	                    #sFB_Conveyor330(iUDT_ConveyorConfiguration := #iUDT_Configuration."330".Conveyor,
	                                     idi_PECEoSDistance := #iUDT_Configuration."330".PEC_Eos.Distance,
	                                     idi_PECBoSDistance := 0,
	                                     ii_ExternalSpeed := 0,
	                                     ix_SafetyOk := #ix_SafetyOk,
	                                     ix_24vOk := #ix_24vOk,
	                                     ix_400vOk := #ix_400vOk,
	                                     ix_HardwareOk := #ix_HardwareOk,
	                                     ix_PECEoS := #iqUDT_WorkstationStatus."330".PEC_EoS.PEC,
	                                     ix_PECBoS := TRUE,
	                                     ix_ReverseDirection := FALSE,
	                                     ix_ExternalRequestDieBack := FALSE,
	                                     ix_ExternalRequestHold := #sx_LeftExternalRequestHold330,
	                                     ix_ResetEnergySave := FALSE,
	                                     qUDT_HMIStatus => #iqUDT_WorkstationStatus."330".Conveyor,
	                                     qUDT_Status => #iqUDT_WorkstationCommonStatus."330",
	                                     iqUDT_EquipmentControl := #iqUDT_EquipmentControl,
	                                     iqUDT_ConveyorCommand := #iqUDT_WorkstationCommands."330".Conveyor,
	                                     iqUDT_ConveyorInterface := #sUDT_Interface330,
	                                     iqUDT_HandShakeUp := #sUDT_Handshake320,
	                                     iqUDT_HandShake := #sUDT_Handshake330,
	                                     iqUDT_Statistics := #iqUDT_WorkstationStatistics."330".Conveyor);
	                END_REGION

	                REGION MCO

	                    #sFB_MCOConveyLinxAixController330(iUDT_AixConfig := #iUDT_Configuration."330".MCO_M01,
	                                                       iUDT_AixInputsModule := #iUDT_MotorInput330,
	                                                       ix_24vOk := #ix_24vOk,
	                                                       ix_SimulationModeActive := "DB_Memory".Simulation,
	                                                       ii_MotorPositionId := 1,
	                                                       qUDT_HMIStatus => #iqUDT_WorkstationStatus."330".MCO_M01,
	                                                       iqUDT_AixOutputsModule := #iqUDT_MotorOutput330,
	                                                       iqUDT_ConveyorInterface := #sUDT_Interface330,
	                                                       iqUDT_MCOStatistics := #iqUDT_WorkstationStatistics."330".MCO_M01);
	                END_REGION
	            END_REGION

	            REGION 340

	                REGION Displacement

	                    #sFB_Displacement340(#sUDT_Interface340);

	                END_REGION

	                REGION EOS
	                    #sFB_PEC340(ix_PEC := NOT #iUDT_MotorInput330.AllSensorPortInputs.RightSensor,
	                                iUDT_PECConfiguration := #iUDT_Configuration."340".PEC_Eos,
	                                qx_PECFiltered => #tx_dummy,
	                                qUDT_HMIStatus => #iqUDT_WorkstationStatus."340".PEC_EoS,
	                                iqUDT_ConveyorInterface := #sUDT_Interface340,
	                                iqUDT_PECStatistics := #iqUDT_WorkstationStatistics."340".PEC_EoS);


	                END_REGION


	                REGION Conveyor

	                    #sFB_Conveyor340(iUDT_ConveyorConfiguration := #iUDT_Configuration."340".Conveyor,
	                                     idi_PECEoSDistance := #iUDT_Configuration."340".PEC_Eos.Distance,
	                                     idi_PECBoSDistance := 0,
	                                     ii_ExternalSpeed := 0,
	                                     ix_SafetyOk := #ix_SafetyOk,
	                                     ix_24vOk := #ix_24vOk,
	                                     ix_400vOk := #ix_400vOk,
	                                     ix_HardwareOk := #ix_HardwareOk,
	                                     ix_PECEoS := #iqUDT_WorkstationStatus."340".PEC_EoS.PEC,
	                                     ix_PECBoS := TRUE,
	                                     ix_ReverseDirection := FALSE,
	                                     ix_ExternalRequestDieBack := FALSE,
	                                     ix_ExternalRequestHold := #sx_LeftExternalRequestHold340,
	                                     ix_ResetEnergySave := FALSE,
	                                     qUDT_HMIStatus => #iqUDT_WorkstationStatus."340".Conveyor,
	                                     qUDT_Status => #iqUDT_WorkstationCommonStatus."340",
	                                     iqUDT_EquipmentControl := #iqUDT_EquipmentControl,
	                                     iqUDT_ConveyorCommand := #iqUDT_WorkstationCommands."340".Conveyor,
	                                     iqUDT_ConveyorInterface := #sUDT_Interface340,
	                                     iqUDT_HandShakeUp := #sUDT_Handshake330,
	                                     iqUDT_HandShake := #sUDT_Handshake340,
	                                     iqUDT_Statistics := #iqUDT_WorkstationStatistics."340".Conveyor);
	                END_REGION

	                REGION MCO

	                    #sFB_MCOConveyLinxAixController340(iUDT_AixConfig := #iUDT_Configuration."340".MCO_M01,
	                                                       iUDT_AixInputsModule := #iUDT_MotorInput330,
	                                                       ix_24vOk := #ix_24vOk,
	                                                       ix_SimulationModeActive := "DB_Memory".Simulation,
	                                                       ii_MotorPositionId := 2,
	                                                       qUDT_HMIStatus => #iqUDT_WorkstationStatus."340".MCO_M01,
	                                                       iqUDT_AixOutputsModule := #iqUDT_MotorOutput330,
	                                                       iqUDT_ConveyorInterface := #sUDT_Interface340,
	                                                       iqUDT_MCOStatistics := #iqUDT_WorkstationStatistics."340".MCO_M01);
	                END_REGION
	            END_REGION

	            REGION 350

	                REGION Displacement

	                    #sFB_Displacement350(#sUDT_Interface350);

	                END_REGION

	                REGION EOS
	                    #sFB_PEC350(ix_PEC := NOT #iUDT_MotorInput350.AllSensorPortInputs.LeftSensor,
	                                iUDT_PECConfiguration := #iUDT_Configuration."350".PEC_Eos,
	                                qx_PECFiltered => #tx_dummy,
	                                qUDT_HMIStatus => #iqUDT_WorkstationStatus."350".PEC_EoS,
	                                iqUDT_ConveyorInterface := #sUDT_Interface350,
	                                iqUDT_PECStatistics := #iqUDT_WorkstationStatistics."350".PEC_EoS);

	                END_REGION

	                REGION Conveyor

	                    #sUDT_Handshake350.RTR := #sUDT_Handshake350.RTR OR #iqUDT_WorkstationStatus."350".PEC_EoS.PEC;

	                    #sFB_Conveyor350(iUDT_ConveyorConfiguration := #iUDT_Configuration."350".Conveyor,
	                                     idi_PECEoSDistance := #iUDT_Configuration."350".PEC_Eos.Distance,
	                                     idi_PECBoSDistance := 0,
	                                     ii_ExternalSpeed := 0,
	                                     ix_SafetyOk := #ix_SafetyOk,
	                                     ix_24vOk := #ix_24vOk,
	                                     ix_400vOk := #ix_400vOk,
	                                     ix_HardwareOk := #ix_HardwareOk,
	                                     ix_PECEoS := #iqUDT_WorkstationStatus."350".PEC_EoS.PEC,
	                                     ix_PECBoS := TRUE,
	                                     ix_ReverseDirection := FALSE,
	                                     ix_ExternalRequestDieBack := FALSE,
	                                     ix_ExternalRequestHold := #sx_LeftExternalRequestHold350,
	                                     ix_ResetEnergySave := FALSE,
	                                     qUDT_HMIStatus => #iqUDT_WorkstationStatus."350".Conveyor,
	                                     qUDT_Status => #iqUDT_WorkstationCommonStatus."350",
	                                     iqUDT_EquipmentControl := #iqUDT_EquipmentControl,
	                                     iqUDT_ConveyorCommand := #iqUDT_WorkstationCommands."350".Conveyor,
	                                     iqUDT_ConveyorInterface := #sUDT_Interface350,
	                                     iqUDT_HandShakeUp := #sUDT_Handshake340,
	                                     iqUDT_HandShake := #sUDT_Handshake350,
	                                     iqUDT_Statistics := #iqUDT_WorkstationStatistics."350".Conveyor);
	                END_REGION

	                REGION MCO

	                    #sFB_MCOConveyLinxAixController350(iUDT_AixConfig := #iUDT_Configuration."350".MCO_M01,
	                                                       iUDT_AixInputsModule := #iUDT_MotorInput350,
	                                                       ix_24vOk := #ix_24vOk,
	                                                       ix_SimulationModeActive := "DB_Memory".Simulation,
	                                                       ii_MotorPositionId := 1,
	                                                       qUDT_HMIStatus => #iqUDT_WorkstationStatus."350".MCO_M01,
	                                                       iqUDT_AixOutputsModule := #iqUDT_MotorOutput350,
	                                                       iqUDT_ConveyorInterface := #sUDT_Interface350,
	                                                       iqUDT_MCOStatistics := #iqUDT_WorkstationStatistics."350".MCO_M01);
	                END_REGION
	            END_REGION
	        END_REGION
	    END_IF;
	END_REGION

	REGION 6 - Right station
	    IF #iUDT_Configuration.GlobalConfig.RightStationExists THEN

	        REGION 6.1 - Indexing

	            // Start indexing after request if there are empty stations and no pushout is active
	            IF #iqUDT_CommunicationWES.RightWorkstation.StartIndexing AND #si_RightEmptyStations > 0
	                AND NOT (#sx_RightPushOutActiveStation1
	                OR #sx_RightPushOutActiveStation2
	                OR #sx_RightPushOutActiveStation3
	                OR #sx_RightPushOutActiveStation4
	                OR #sx_RightPushOutActiveStation5) THEN

	                #sx_RightIndexing := TRUE;
	            END_IF;

	            IF NOT #sx_RightIndexing THEN                                      // If there is no indexing in progress

	                #si_RightDestinationC541 := 0;                                // Reset RAT destination
	                #sx_RightExternalRequestHold550 := TRUE;                      // Hold station conveyors
	                #sx_RightExternalRequestHold560 := TRUE;
	                #sx_RightExternalRequestHold570 := TRUE;
	                #sx_RightExternalRequestHold580 := TRUE;
	                #sx_RightExternalRequestHold590 := TRUE;

	            ELSE

	                IF #sR_TRIG_PEC540.Q AND #si_RightEmptyStations > 0 THEN       //Count down empty stations after diverting a tote into station
	                    #si_RightEmptyStations -= 1;
	                END_IF;

	                #si_RightDestinationC541 := 1;                               // Set RAT destination
	                #sx_RightExternalRequestHold550 := FALSE;                    // Release hold of station conveyors
	                #sx_RightExternalRequestHold560 := FALSE;
	                #sx_RightExternalRequestHold570 := FALSE;
	                #sx_RightExternalRequestHold580 := FALSE;
	                #sx_RightExternalRequestHold590 := FALSE;

	                IF                                                           //End indexing when all totes are on position
	                    NOT #iqUDT_WorkstationStatus."550".PEC_EoS.PEC
	                    AND NOT #iqUDT_WorkstationStatus."560".PEC_EoS.PEC
	                    AND NOT #iqUDT_WorkstationStatus."570".PEC_EoS.PEC
	                    AND NOT #iqUDT_WorkstationStatus."580".PEC_EoS.PEC
	                    AND NOT #iqUDT_WorkstationStatus."590".PEC_EoS.PEC
	                    AND NOT (#sUDT_Interface550.ActualSpeed > 0) THEN

	                    #sx_RightIndexing := FALSE;

	                END_IF;
	            END_IF;

	        END_REGION

	        REGION 6.2 - Push Out

	            REGION 6.2.0 - Pushout conveyors hold
	                IF #sFB_TimerOnOffDelay_Hold710.qx_DelayedSignal THEN
	                    #sx_RightExternalRequestHold710 := TRUE;
	                END_IF;

	                IF #sFB_TimerOnOffDelay_Hold720.qx_DelayedSignal THEN
	                    #sx_RightExternalRequestHold720 := TRUE;
	                END_IF;

	                IF #sFB_TimerOnOffDelay_Hold730.qx_DelayedSignal THEN
	                    #sx_RightExternalRequestHold730 := TRUE;
	                END_IF;

	                IF #sFB_TimerOnOffDelay_Hold740.qx_DelayedSignal THEN
	                    #sx_RightExternalRequestHold740 := TRUE;
	                END_IF;

	                IF #sFB_TimerOnOffDelay_Hold750.qx_DelayedSignal THEN
	                    #sx_RightExternalRequestHold750 := TRUE;
	                END_IF;
	            END_REGION

	            REGION 6.2.1 - Push Out Station 1

	                // Start automatic pushout after request if there is no indexing procedure and a tote is present on first station
	                IF #iqUDT_CommunicationWES.RightWorkstation.Station1.ReadyForPush AND NOT #sx_RightIndexing
	                    AND NOT #iqUDT_WorkstationStatus."590".PEC_EoS.PEC THEN

	                    #sx_RightPushOutActiveStation1 := TRUE;
	                END_IF;

	                IF #sx_RightPushOutActiveStation1 THEN                         //release hold
	                    #sx_RightExternalRequestHold590 := FALSE;

	                    IF #sFB_RightAngledTransfer611.qx_ExternalSendRequestB THEN    //after tote is already on RAT, hold the conveyor and end pushout procedure
	                        #sx_RightExternalRequestHold590 := TRUE;
	                        #sx_RightPushOutActiveStation1 := FALSE;
	                    END_IF;
	                END_IF;

	            END_REGION

	            REGION 6.2.2 - Push Out station 2

	                IF #iqUDT_CommunicationWES.RightWorkstation.Station2.ReadyForPush THEN        //set pushout to active after request
	                    #sx_RightPushOutActiveStation2 := TRUE;
	                END_IF;

	                IF #sx_RightPushOutActiveStation2                               // After station is empty and tote has been detected on pushout conveyor release holds
	                    AND #iqUDT_WorkstationStatus."580".PEC_EoS.PEC
	                    AND #sFB_TimerOnOffDelay_Detect740.qx_DelayedSignal THEN

	                    #sx_RightExternalRequestHold740 := FALSE;
	                    #sx_RightExternalRequestHold750 := FALSE;

	                    FILL_BLK(IN := 0,                                             //clear tracking
	                             COUNT := REAL_TO_ULINT(DINT_TO_REAL(#iUDT_Configuration."580".Conveyor.Common.Length) * #cr_ClearTrackingModifier),
	                             OUT => #sa_TrackingArray580[0]);

	                    #sx_RightPushOutActiveStation2 := FALSE;                       //end pushout procedure

	                END_IF;


	            END_REGION

	            REGION 6.2.3 - Push Out station 3

	                IF #iqUDT_CommunicationWES.RightWorkstation.Station3.ReadyForPush THEN          //set pushout to active after request
	                    #sx_RightPushOutActiveStation3 := TRUE;
	                END_IF;

	                IF #sx_RightPushOutActiveStation3
	                    AND #iqUDT_WorkstationStatus."570".PEC_EoS.PEC
	                    AND #sFB_TimerOnOffDelay_Detect730.qx_DelayedSignal THEN                // After station is empty and tote has been detected on pushout conveyor release holds

	                    #sx_RightExternalRequestHold730 := FALSE;
	                    #sx_RightExternalRequestHold740 := FALSE;
	                    #sx_RightExternalRequestHold750 := FALSE;

	                    FILL_BLK(IN := 0,                                                         //clear tracking
	                             COUNT := REAL_TO_ULINT(DINT_TO_REAL(#iUDT_Configuration."570".Conveyor.Common.Length) * #cr_ClearTrackingModifier),
	                             OUT => #sa_TrackingArray570[0]);

	                    #sx_RightPushOutActiveStation3 := FALSE;                              //end pushout procedure

	                END_IF;
	            END_REGION

	            REGION 6.2.4 - Push Out station 4

	                IF #iqUDT_CommunicationWES.RightWorkstation.Station4.ReadyForPush THEN              //set pushout to active after request
	                    #sx_RightPushOutActiveStation4 := TRUE;
	                END_IF;

	                IF #sx_RightPushOutActiveStation4
	                    AND #iqUDT_WorkstationStatus."560".PEC_EoS.PEC
	                    AND #sFB_TimerOnOffDelay_Detect720.qx_DelayedSignal THEN                // After station is empty and tote has been detected on pushout conveyor release holds

	                    #sx_RightExternalRequestHold720 := FALSE;
	                    #sx_RightExternalRequestHold730 := FALSE;
	                    #sx_RightExternalRequestHold740 := FALSE;
	                    #sx_RightExternalRequestHold750 := FALSE;

	                    FILL_BLK(IN := 0,                                                      //clear tracking
	                             COUNT := REAL_TO_ULINT(DINT_TO_REAL(#iUDT_Configuration."560".Conveyor.Common.Length) * #cr_ClearTrackingModifier),
	                             OUT => #sa_TrackingArray560[0]);

	                    #sx_RightPushOutActiveStation4 := FALSE;                          //end pushout procedure

	                END_IF;

	            END_REGION

	            REGION 6.2.5 - Push Out station 5

	                IF #iqUDT_CommunicationWES.RightWorkstation.Station5.ReadyForPush THEN          //set pushout to active after request
	                    #sx_RightPushOutActiveStation5 := TRUE;
	                END_IF;

	                IF #sx_RightPushOutActiveStation5
	                    AND #iqUDT_WorkstationStatus."550".PEC_EoS.PEC
	                    AND #sFB_TimerOnOffDelay_Detect710.qx_DelayedSignal THEN                // After station is empty and tote has been detected on pushout conveyor release holds

	                    #sx_RightExternalRequestHold710 := FALSE;
	                    #sx_RightExternalRequestHold720 := FALSE;
	                    #sx_RightExternalRequestHold730 := FALSE;
	                    #sx_RightExternalRequestHold740 := FALSE;
	                    #sx_RightExternalRequestHold750 := FALSE;

	                    FILL_BLK(IN := 0,                                            //clear tracking
	                             COUNT := REAL_TO_ULINT(DINT_TO_REAL(#iUDT_Configuration."550".Conveyor.Common.Length) * #cr_ClearTrackingModifier),
	                             OUT => #sa_TrackingArray550[0]);

	                    #sx_RightPushOutActiveStation5 := FALSE;                      //end pushout procedure
	                END_IF;

	            END_REGION

	        END_REGION

	        REGION 6.3 WES Communication
	            REGION 6.3.1 Lost track error

	                IF NOT #sx_RightIndexing
	                    AND NOT #sx_RightPushOutActiveStation1
	                    AND #sa_TrackingArray590[30] >= 1000
	                    AND #iqUDT_WorkstationStatus."590".PEC_EoS.PEC THEN
	                    #iqUDT_CommunicationWES.RightWorkstation.Station1.Error := TRUE;
	                END_IF;

	                IF NOT #sx_RightIndexing
	                    AND NOT #sx_RightPushOutActiveStation2
	                    AND #sa_TrackingArray580[30] >= 1000
	                    AND #iqUDT_WorkstationStatus."580".PEC_EoS.PEC THEN
	                    #iqUDT_CommunicationWES.RightWorkstation.Station2.Error := TRUE;
	                END_IF;

	                IF NOT #sx_RightIndexing
	                    AND NOT #sx_RightPushOutActiveStation3
	                    AND #sa_TrackingArray570[30] >= 1000
	                    AND #iqUDT_WorkstationStatus."570".PEC_EoS.PEC THEN
	                    #iqUDT_CommunicationWES.RightWorkstation.Station3.Error := TRUE;
	                END_IF;

	                IF NOT #sx_RightIndexing
	                    AND NOT #sx_RightPushOutActiveStation4
	                    AND #sa_TrackingArray560[30] >= 1000
	                    AND #iqUDT_WorkstationStatus."560".PEC_EoS.PEC THEN
	                    #iqUDT_CommunicationWES.RightWorkstation.Station4.Error := TRUE;
	                END_IF;

	                IF NOT #sx_RightIndexing
	                    AND NOT #sx_RightPushOutActiveStation5
	                    AND #sa_TrackingArray550[30] >= 1000
	                    AND #iqUDT_WorkstationStatus."550".PEC_EoS.PEC THEN
	                    #iqUDT_CommunicationWES.RightWorkstation.Station5.Error := TRUE;
	                END_IF;

	            END_REGION

	            REGION 6.3.2 Reset lost errors

	                IF #iqUDT_EquipmentControl.Command.Reset                   // Reset command received
	                THEN
	                    #iqUDT_CommunicationWES.RightWorkstation.Station1.Error := FALSE;
	                    #iqUDT_CommunicationWES.RightWorkstation.Station2.Error := FALSE;
	                    #iqUDT_CommunicationWES.RightWorkstation.Station3.Error := FALSE;
	                    #iqUDT_CommunicationWES.RightWorkstation.Station4.Error := FALSE;
	                    #iqUDT_CommunicationWES.RightWorkstation.Station5.Error := FALSE;
	                END_IF;

	            END_REGION

	            REGION 6.3.3 GIN at station
	                IF NOT #sx_RightIndexing THEN
	                    IF NOT #sx_RightPushOutActiveStation1 THEN
	                        #iqUDT_CommunicationWES.RightWorkstation.Station1.Gin := #sa_TrackingArray590[23];
	                    END_IF;
	                    #iqUDT_CommunicationWES.RightWorkstation.Station2.Gin := #sa_TrackingArray580[23];
	                    #iqUDT_CommunicationWES.RightWorkstation.Station3.Gin := #sa_TrackingArray570[23];
	                    #iqUDT_CommunicationWES.RightWorkstation.Station4.Gin := #sa_TrackingArray560[23];
	                    #iqUDT_CommunicationWES.RightWorkstation.Station5.Gin := #sa_TrackingArray550[23];
	                END_IF;
	            END_REGION

	            REGION 6.3.4 Barcode at station
	                //Write barcode to WES

	                IF (#iqUDT_CommunicationWES.RightWorkstation.Station1.Gin > 0) AND (#iqUDT_CommunicationWES.RightWorkstation.Station1.Gin < 10000) THEN
	                    #iqUDT_CommunicationWES.RightWorkstation.Station1.Barcode := "DB_GIN".GIN[#iqUDT_CommunicationWES.RightWorkstation.Station1.Gin].WES.Barcode;
	                ELSE
	                    #iqUDT_CommunicationWES.RightWorkstation.Station1.Barcode := '          ';
	                END_IF;

	                IF (#iqUDT_CommunicationWES.RightWorkstation.Station2.Gin > 0) AND (#iqUDT_CommunicationWES.RightWorkstation.Station2.Gin < 10000) THEN
	                    #iqUDT_CommunicationWES.RightWorkstation.Station2.Barcode := "DB_GIN".GIN[#iqUDT_CommunicationWES.RightWorkstation.Station2.Gin].WES.Barcode;
	                ELSE
	                    #iqUDT_CommunicationWES.RightWorkstation.Station2.Barcode := '          ';
	                END_IF;

	                IF (#iqUDT_CommunicationWES.RightWorkstation.Station3.Gin > 0) AND (#iqUDT_CommunicationWES.RightWorkstation.Station3.Gin < 10000) THEN
	                    #iqUDT_CommunicationWES.RightWorkstation.Station3.Barcode := "DB_GIN".GIN[#iqUDT_CommunicationWES.RightWorkstation.Station3.Gin].WES.Barcode;
	                ELSE
	                    #iqUDT_CommunicationWES.RightWorkstation.Station3.Barcode := '          ';
	                END_IF;

	                IF (#iqUDT_CommunicationWES.RightWorkstation.Station4.Gin > 0) AND (#iqUDT_CommunicationWES.RightWorkstation.Station4.Gin < 10000) THEN
	                    #iqUDT_CommunicationWES.RightWorkstation.Station4.Barcode := "DB_GIN".GIN[#iqUDT_CommunicationWES.RightWorkstation.Station4.Gin].WES.Barcode;
	                ELSE
	                    #iqUDT_CommunicationWES.RightWorkstation.Station4.Barcode := '          ';
	                END_IF;

	                IF (#iqUDT_CommunicationWES.RightWorkstation.Station5.Gin > 0) AND (#iqUDT_CommunicationWES.RightWorkstation.Station5.Gin < 10000) THEN
	                    #iqUDT_CommunicationWES.RightWorkstation.Station5.Barcode := "DB_GIN".GIN[#iqUDT_CommunicationWES.RightWorkstation.Station5.Gin].WES.Barcode;
	                ELSE
	                    #iqUDT_CommunicationWES.RightWorkstation.Station5.Barcode := '          ';
	                END_IF;

	            END_REGION


	        END_REGION

	        REGION 6.4 - Function block calls
	            REGION 510

	                REGION Displacement

	                    #sFB_Displacement510(#sUDT_Interface510);

	                END_REGION

	                REGION Conveyor

	                    #sFB_Conveyor510(iUDT_ConveyorConfiguration := #iUDT_Configuration."510".Conveyor,
	                                     idi_PECEoSDistance := 0,
	                                     idi_PECBoSDistance := 0,
	                                     ii_ExternalSpeed := 0,
	                                     ix_SafetyOk := #ix_SafetyOk,
	                                     ix_24vOk := #ix_24vOk,
	                                     ix_400vOk := #ix_400vOk,
	                                     ix_HardwareOk := #ix_HardwareOk,
	                                     ix_PECEoS := TRUE,
	                                     ix_PECBoS := TRUE,
	                                     ix_ReverseDirection := FALSE,
	                                     ix_ExternalRequestDieBack := FALSE,
	                                     ix_ExternalRequestHold := FALSE,
	                                     ix_ResetEnergySave := FALSE,
	                                     qUDT_HMIStatus => #iqUDT_WorkstationStatus."510".Conveyor,
	                                     qUDT_Status => #iqUDT_WorkstationCommonStatus."510",
	                                     iqUDT_EquipmentControl := #iqUDT_EquipmentControl,
	                                     iqUDT_ConveyorCommand := #iqUDT_WorkstationCommands."510".Conveyor,
	                                     iqUDT_ConveyorInterface := #sUDT_Interface510,
	                                     iqUDT_HandShakeUp := #sUDT_HandshakeUp020,
	                                     iqUDT_HandShake := #sUDT_Handshake510,
	                                     iqUDT_Statistics := #iqUDT_WorkstationStatistics."510".Conveyor);
	                END_REGION

	                REGION MCO

	                    #sFB_MCOConveyLinxAixController510(iUDT_AixConfig := #iUDT_Configuration."510".MCO_M01,
	                                                       iUDT_AixInputsModule := #iUDT_MotorInput510,
	                                                       ix_24vOk := #ix_24vOk,
	                                                       ix_SimulationModeActive := "DB_Memory".Simulation,
	                                                       ii_MotorPositionId := 1,
	                                                       qUDT_HMIStatus => #iqUDT_WorkstationStatus."510".MCO_M01,
	                                                       iqUDT_AixOutputsModule := #iqUDT_MotorOutput510,
	                                                       iqUDT_ConveyorInterface := #sUDT_Interface510,
	                                                       iqUDT_MCOStatistics := #iqUDT_WorkstationStatistics."510".MCO_M01);
	                END_REGION
	            END_REGION

	            REGION 520

	                REGION Displacement

	                    #sFB_Displacement520(#sUDT_Interface520);

	                END_REGION

	                REGION Tracking
	                    #sFB_Tracking520(iUDT_ConveyorCommonConfiguration := #iUDT_Configuration."520".Conveyor.Common,
	                                     iqa_TrackingData := #sa_TrackingArray520,
	                                     iqUDT_ConveyorInterface := #sUDT_Interface520,
	                                     iqUDT_HandshakeUp := #sUDT_Handshake510,
	                                     iqUDT_Handshake := #sUDT_Handshake520);

	                END_REGION


	                REGION EOS

	                    #sFB_PECUpdate520(iUDT_PECUpdateConfiguration := #iUDT_Configuration."520".PEC_Eos,
	                                      iUDT_ConveyorCommonConfiguration := #iUDT_Configuration."520".Conveyor.Common,
	                                      ix_PEC := #iUDT_MotorInput520.AllSensorPortInputs.LeftSensor,
	                                      ix_TeachingMode := FALSE,
	                                      qUDT_Status => #iqUDT_WorkstationStatus."520".PEC_EoS,
	                                      qi_GINwrite => #ti_dummy,
	                                      qx_PECFiltered => #tx_dummy,
	                                      iqUDT_ConveyorInterface := #sUDT_Interface520,
	                                      iqUDT_UnknownGINRange := #iqUDT_UnknownGINRange,
	                                      iqUDT_FifoHeader := "DB_FIFOLostGIN".Header,
	                                      iqUDT_Statistics := #iqUDT_WorkstationStatistics."520".PEC_EoS,
	                                      iqa_TrackingData := #sa_TrackingArray520,
	                                      iqa_FifoData := "DB_FIFOLostGIN".Data);

	                END_REGION

	                REGION Conveyor

	                    #sFB_Conveyor520(iUDT_ConveyorConfiguration := #iUDT_Configuration."520".Conveyor,
	                                     idi_PECEoSDistance := #iUDT_Configuration."520".PEC_Eos.Distance,
	                                     idi_PECBoSDistance := 0,
	                                     ii_ExternalSpeed := 0,
	                                     ix_SafetyOk := #ix_SafetyOk,
	                                     ix_24vOk := #ix_24vOk,
	                                     ix_400vOk := #ix_400vOk,
	                                     ix_HardwareOk := #ix_HardwareOk,
	                                     ix_PECEoS := #iqUDT_WorkstationStatus."520".PEC_EoS.PEC,
	                                     ix_PECBoS := TRUE,
	                                     ix_ReverseDirection := FALSE,
	                                     ix_ExternalRequestDieBack := FALSE,
	                                     ix_ExternalRequestHold := FALSE,
	                                     ix_ResetEnergySave := FALSE,
	                                     qUDT_HMIStatus => #iqUDT_WorkstationStatus."520".Conveyor,
	                                     qUDT_Status => #iqUDT_WorkstationCommonStatus."520",
	                                     iqUDT_EquipmentControl := #iqUDT_EquipmentControl,
	                                     iqUDT_ConveyorCommand := #iqUDT_WorkstationCommands."520".Conveyor,
	                                     iqUDT_ConveyorInterface := #sUDT_Interface520,
	                                     iqUDT_HandShakeUp := #sUDT_Handshake510,
	                                     iqUDT_HandShake := #sUDT_Handshake520,
	                                     iqUDT_Statistics := #iqUDT_WorkstationStatistics."520".Conveyor);
	                END_REGION

	                REGION MCO

	                    #sFB_MCOConveyLinxAixController520(iUDT_AixConfig := #iUDT_Configuration."520".MCO_M01,
	                                                       iUDT_AixInputsModule := #iUDT_MotorInput520,
	                                                       ix_24vOk := #ix_24vOk,
	                                                       ix_SimulationModeActive := "DB_Memory".Simulation,
	                                                       ii_MotorPositionId := 1,
	                                                       qUDT_HMIStatus => #iqUDT_WorkstationStatus."520".MCO_M01,
	                                                       iqUDT_AixOutputsModule := #iqUDT_MotorOutput520,
	                                                       iqUDT_ConveyorInterface := #sUDT_Interface520,
	                                                       iqUDT_MCOStatistics := #iqUDT_WorkstationStatistics."520".MCO_M01);
	                END_REGION
	            END_REGION

	            REGION 530

	                REGION Displacement

	                    #sFB_Displacement530(#sUDT_Interface530);

	                END_REGION

	                REGION Tracking

	                    #sFB_Tracking530(iUDT_ConveyorCommonConfiguration := #iUDT_Configuration."530".Conveyor.Common,
	                                     iqa_TrackingData := #sa_TrackingArray530,
	                                     iqUDT_ConveyorInterface := #sUDT_Interface530,
	                                     iqUDT_HandshakeUp := #sUDT_Handshake520,
	                                     iqUDT_Handshake := #sUDT_Handshake530);

	                END_REGION

	                REGION EOS

	                    #sFB_PECUpdate530(iUDT_PECUpdateConfiguration := #iUDT_Configuration."530".PEC_Eos,
	                                      iUDT_ConveyorCommonConfiguration := #iUDT_Configuration."530".Conveyor.Common,
	                                      ix_PEC := #iUDT_MotorInput520.AllSensorPortInputs.RightSensor,
	                                      ix_TeachingMode := FALSE,
	                                      qUDT_Status => #iqUDT_WorkstationStatus."530".PEC_EoS,
	                                      qi_GINwrite => #ti_dummy,
	                                      qx_PECFiltered => #tx_dummy,
	                                      iqUDT_ConveyorInterface := #sUDT_Interface530,
	                                      iqUDT_UnknownGINRange := #iqUDT_UnknownGINRange,
	                                      iqUDT_FifoHeader := "DB_FIFOLostGIN".Header,
	                                      iqUDT_Statistics := #iqUDT_WorkstationStatistics."530".PEC_EoS,
	                                      iqa_TrackingData := #sa_TrackingArray530,
	                                      iqa_FifoData := "DB_FIFOLostGIN".Data);

	                END_REGION

	                REGION Scanner

	                    // #sFB_CognexCamera260_530(iUDT_CognexDM260_IN       := #iUDT_ScannerInput530,
	                    //                          iUDT_EquipmentControl:=#iqUDT_EquipmentControl,
	                    //                          ix_Trigger                := #sa_TrackingArray_130[38]>1000,
	                    //                          qUDT_CognexDM260_OUT      => #qUDT_ScannerOutput530,
	                    //                          qs_Barcode                => #ts_Barcode530,
	                    //                          qw_RetVal                 => #tw_dummy);00
	                    //

	                    // IF #sa_TrackingArray_530[38] > 0 THEN
	                    //     #ti_GIN := #sa_TrackingArray_530[38];
	                    //     "DB_GIN".GIN[#ti_GIN].WES.Barcode := #ts_Barcode530;
	                    // END_IF;
	                    //


	                    #sFB_DataLogicBlade200_530(iUDT_DataLogic := #iUDT_ScannerInput530,
	                                               ix_trigger := #sa_TrackingArray530[27] > 0,
	                                               qUDT_DataLogic => #qudt_ScannerOutput530,
	                                               qs_Barcode => #ts_Barcode530,
	                                               qw_RetVal => #tw_dummy,
	                                               iqUDT_EquipmentControl := #iqUDT_EquipmentControl);

	                    IF #sa_TrackingArray530[47] > 0 THEN
	                        #ti_GIN530 := #sa_TrackingArray530[47];
	                        "DB_GIN".GIN[#ti_GIN530].WES.Barcode := #ts_Barcode530;
	                    END_IF;

	                END_REGION

	                REGION Conveyor

	                    #sUDT_Handshake530.RTR := #iqUDT_WorkstationStatus."530".PEC_EoS.PEC OR
	                    (#iqUDT_WorkstationStatus."540".PEC_EoS.PEC AND #sUDT_Interface540.ActualSpeed <> 0);

	                    #sFB_Conveyor530(iUDT_ConveyorConfiguration := #iUDT_Configuration."530".Conveyor,
	                                     idi_PECEoSDistance := #iUDT_Configuration."530".PEC_Eos.Distance,
	                                     idi_PECBoSDistance := 0,
	                                     ii_ExternalSpeed := 0,
	                                     ix_SafetyOk := #ix_SafetyOk,
	                                     ix_24vOk := #ix_24vOk,
	                                     ix_400vOk := #ix_400vOk,
	                                     ix_HardwareOk := #ix_HardwareOk,
	                                     ix_PECEoS := #iqUDT_WorkstationStatus."530".PEC_EoS.PEC,
	                                     ix_PECBoS := TRUE,
	                                     ix_ReverseDirection := FALSE,
	                                     ix_ExternalRequestDieBack := FALSE,
	                                     ix_ExternalRequestHold := FALSE,
	                                     ix_ResetEnergySave := FALSE,
	                                     qUDT_HMIStatus => #iqUDT_WorkstationStatus."530".Conveyor,
	                                     qUDT_Status => #iqUDT_WorkstationCommonStatus."530",
	                                     iqUDT_EquipmentControl := #iqUDT_EquipmentControl,
	                                     iqUDT_ConveyorCommand := #iqUDT_WorkstationCommands."530".Conveyor,
	                                     iqUDT_ConveyorInterface := #sUDT_Interface530,
	                                     iqUDT_HandShakeUp := #sUDT_Handshake520,
	                                     iqUDT_HandShake := #sUDT_Handshake530,
	                                     iqUDT_Statistics := #iqUDT_WorkstationStatistics."530".Conveyor);
	                END_REGION

	                REGION MCO

	                    #sFB_MCOConveyLinxAixController530(iUDT_AixConfig := #iUDT_Configuration."530".MCO_M01,
	                                                       iUDT_AixInputsModule := #iUDT_MotorInput520,
	                                                       ix_24vOk := #ix_24vOk,
	                                                       ix_SimulationModeActive := "DB_Memory".Simulation,
	                                                       ii_MotorPositionId := 2,
	                                                       qUDT_HMIStatus => #iqUDT_WorkstationStatus."530".MCO_M01,
	                                                       iqUDT_AixOutputsModule := #iqUDT_MotorOutput520,
	                                                       iqUDT_ConveyorInterface := #sUDT_Interface530,
	                                                       iqUDT_MCOStatistics := #iqUDT_WorkstationStatistics."530".MCO_M01);
	                END_REGION

	            END_REGION

	            REGION 540

	                REGION Displacement

	                    #sFB_Displacement540(#sUDT_Interface540);

	                END_REGION

	                REGION MCO

	                    #sFB_MCOConveyLinxAixController540(iUDT_AixConfig := #iUDT_Configuration."540".MCO_M01,
	                                                       iUDT_AixInputsModule := #iUDT_MotorInput540,
	                                                       ii_PositionSetpoint := #iqUDT_RATPositioning540.Lower.EndPosition,
	                                                       ix_24vOk := #ix_24vOk,
	                                                       ix_SimulationModeActive := "DB_Memory".Simulation,
	                                                       ii_MotorPositionId := 1,
	                                                       ix_StartPositioning := #iqUDT_RATPositioning540.Lower.Start,
	                                                       ix_ResetPosition := #iqUDT_RATPositioning540.Lower.ResetPosition,
	                                                       qUDT_HMIStatus => #iqUDT_WorkstationStatus."540".MCO_M01,
	                                                       qx_Positioned => #iqUDT_RATPositioning540.Lower.Done,
	                                                       iqUDT_AixOutputsModule := #iqUDT_MotorOutput540,
	                                                       iqUDT_ConveyorInterface := #sUDT_Interface540,
	                                                       iqUDT_MCOStatistics := #iqUDT_WorkstationStatistics."540".MCO_M01);
	                END_REGION
	            END_REGION

	            REGION 541

	                REGION Displacement

	                    #sFB_Displacement541(#sUDT_Interface541);

	                END_REGION

	                REGION RAT
	                    #sUDT_Handshake541.RTR := #sx_RightIndexing AND
	                    (#iqUDT_WorkstationStatus."550".PEC_EoS.PEC AND #sUDT_Interface550.ActualSpeed <> 0);

	                    #sFB_RightAngledTransfer541(iUDT_Configuration := #iUDT_Configuration."541".RightAngledTransfer,
	                                                iUDT_LowerConveyorConfiguration := #iUDT_Configuration."540".Conveyor,
	                                                iUDT_UpperConveyorConfiguration := #iUDT_Configuration."541".Conveyor,
	                                                iUDT_PECConfiguration := #iUDT_Configuration."540".PEC_EoS,
	                                                ii_DestinationA := #si_RightDestinationC541,
	                                                ii_DestinationB := 0,
	                                                ii_DestinationC := 0,
	                                                ii_DestinationD := 0,
	                                                ix_HardwareOk := #ix_HardwareOk,
	                                                ix_400vOk := #ix_400vOk,
	                                                ix_24vOk := #ix_24vOk,
	                                                ix_SafetyOk := #ix_SafetyOk,
	                                                ix_AirPressureOk := #ix_AirPressureOk,
	                                                ix_SectionIsDown := #ix_SectionIsDown541,
	                                                ix_SectionIsUp := #ix_SectionIsUp541,
	                                                ix_ConveyorAAuto := #iqUDT_WorkstationCommonStatus."530".AutoON,
	                                                ix_ConveyorBAuto := false,
	                                                ix_ConveyorCAuto := false,
	                                                ix_ConveyorDAuto := false,
	                                                ix_PEC := #iUDT_MotorInput540.AllSensorPortInputs.LeftSensor,
	                                                ix_ExternalReceiveRequestA := NOT #iqUDT_WorkstationStatus."530".PEC_EoS.PEC,
	                                                ix_ExternalReceiveRequestB := FALSE,
	                                                ix_ExternalReceiveRequestC := FALSE,
	                                                ix_ExternalReceiveRequestD := FALSE,
	                                                ix_PECInfeedA := #iqUDT_WorkstationStatus."530".PEC_EoS.PEC,
	                                                qUDT_HMIRATStatus => #iqUDT_WorkstationStatus."541".RightAngledTransfer,
	                                                qUDT_HMIConveyorStatus => #iqUDT_WorkstationStatus."540".Conveyor,
	                                                qUDT_HMIPECStatus => #iqUDT_WorkstationStatus."540".PEC_EoS,
	                                                qUDT_RATStatus => #iqUDT_WorkstationCommonStatus."541",
	                                                qUDT_ConveyorStatus => #iqUDT_WorkstationCommonStatus."540",
	                                                qx_PopupControl => #qx_PopupControl541,
	                                                qx_ExternalSendRequestA => #tx_dummy,
	                                                qx_ExternalSendRequestB => #tx_dummy,
	                                                qx_ExternalSendRequestC => #tx_dummy,
	                                                qx_ExternalSendRequestD => #tx_dummy,
	                                                iqUDT_EquipmentControl := #iqUDT_EquipmentControl,
	                                                iqUDT_RATCommand := #iqUDT_WorkstationCommands."541".RightAngledTransfer,
	                                                iqUDT_ConveyorCommand := #iqUDT_WorkstationCommands."540".Conveyor,
	                                                iqUDT_RATStatistics := #iqUDT_WorkstationStatistics."541".RightAngledTransfer,
	                                                iqUDT_ConveyorStatistics := #iqUDT_WorkstationStatistics."540".Conveyor,
	                                                iqUDT_PECStatistics := #iqUDT_WorkstationStatistics."540".PEC_EoS,
	                                                iqUDT_HandShakeConveyorA := #sUDT_Handshake530,
	                                                iqUDT_HandShakeConveyorB := #sUDT_Handshake540,
	                                                iqUDT_HandShakeConveyorC := #tUDT_DummyConveyorHandshake,
	                                                iqUDT_HandShakeConveyorD := #sUDT_Handshake541,
	                                                iqUDT_LowerConveyorInterface := #sUDT_Interface540,
	                                                iqUDT_UpperConveyorInterface := #sUDT_Interface541,
	                                                iqUDT_RATPositioning := #iqUDT_RATPositioning540,
	                                                iqUDT_BladeStopEoSInterface := #tUDT_DummyBladeStop,
	                                                iqUDT_BladeStopBoSInterface := #tUDT_DummyBladeStop);

	                END_REGION

	                REGION MCO

	                    #sFB_MCOConveyLinxAixController541(iUDT_AixConfig := #iUDT_Configuration."541".MCO_M01,
	                                                       iUDT_AixInputsModule := #iUDT_MotorInput540,
	                                                       ix_24vOk := #ix_24vOk,
	                                                       ix_SimulationModeActive := "DB_Memory".Simulation,
	                                                       ii_MotorPositionId := 2,
	                                                       qUDT_HMIStatus => #iqUDT_WorkstationStatus."541".MCO_M01,
	                                                       iqUDT_AixOutputsModule := #iqUDT_MotorOutput540,
	                                                       iqUDT_ConveyorInterface := #sUDT_Interface541,
	                                                       iqUDT_MCOStatistics := #iqUDT_WorkstationStatistics."541".MCO_M01);
	                END_REGION

	            END_REGION

	            REGION 550

	                REGION Displacement

	                    #sFB_Displacement550(#sUDT_Interface550);

	                END_REGION

	                REGION Tracking

	                    #sFB_Tracking550(iUDT_ConveyorCommonConfiguration := #iUDT_Configuration."550".Conveyor.Common,
	                                     iqa_TrackingData := #sa_TrackingArray550,
	                                     iqUDT_ConveyorInterface := #sUDT_Interface550,
	                                     iqUDT_HandshakeUp := #sUDT_Handshake541,
	                                     iqUDT_Handshake := #sUDT_Handshake550);
	                END_REGION

	                REGION EOS

	                    #sFB_PECUpdate550(iUDT_PECUpdateConfiguration := #iUDT_Configuration."550".PEC_Eos,
	                                      iUDT_ConveyorCommonConfiguration := #iUDT_Configuration."550".Conveyor.Common,
	                                      ix_PEC := NOT #iUDT_MotorInput550.AllSensorPortInputs.LeftSensor,
	                                      ix_TeachingMode := FALSE,
	                                      qUDT_Status => #iqUDT_WorkstationStatus."550".PEC_EoS,
	                                      qi_GINwrite => #ti_dummy,
	                                      qx_PECFiltered => #tx_dummy,
	                                      iqa_TrackingData := #sa_TrackingArray550,
	                                      iqUDT_ConveyorInterface := #sUDT_Interface550,
	                                      iqUDT_UnknownGINRange := #iqUDT_UnknownGINRange,
	                                      iqUDT_FifoHeader := "DB_FIFOLostGIN".Header,
	                                      iqa_FifoData := "DB_FIFOLostGIN".Data,
	                                      iqUDT_Statistics := #iqUDT_WorkstationStatistics."550".PEC_EoS);

	                END_REGION

	                REGION Conveyor

	                    #sUDT_Handshake550.RTR := #sx_RightIndexing AND
	                    ((#iqUDT_WorkstationStatus."560".PEC_EoS.PEC AND #sUDT_Interface560.ActualSpeed <> 0) OR #iqUDT_WorkstationStatus."550".PEC_EoS.PEC);

	                    #sFB_Conveyor550(iUDT_ConveyorConfiguration := #iUDT_Configuration."550".Conveyor,
	                                     idi_PECEoSDistance := #iUDT_Configuration."550".PEC_Eos.Distance,
	                                     idi_PECBoSDistance := 0,
	                                     ii_ExternalSpeed := 0,
	                                     ix_SafetyOk := #ix_SafetyOk,
	                                     ix_24vOk := #ix_24vOk,
	                                     ix_400vOk := #ix_400vOk,
	                                     ix_HardwareOk := #ix_HardwareOk,
	                                     ix_PECEoS := #iqUDT_WorkstationStatus."550".PEC_EoS.PEC,
	                                     ix_PECBoS := TRUE,
	                                     ix_ReverseDirection := FALSE,
	                                     ix_ExternalRequestDieBack := FALSE,
	                                     ix_ExternalRequestHold := #sx_RightExternalRequestHold550,
	                                     ix_ResetEnergySave := FALSE,
	                                     qUDT_HMIStatus => #iqUDT_WorkstationStatus."550".Conveyor,
	                                     qUDT_Status => #iqUDT_WorkstationCommonStatus."550",
	                                     iqUDT_EquipmentControl := #iqUDT_EquipmentControl,
	                                     iqUDT_ConveyorCommand := #iqUDT_WorkstationCommands."550".Conveyor,
	                                     iqUDT_ConveyorInterface := #sUDT_Interface550,
	                                     iqUDT_HandShakeUp := #sUDT_Handshake541,
	                                     iqUDT_HandShake := #sUDT_Handshake550,
	                                     iqUDT_Statistics := #iqUDT_WorkstationStatistics."550".Conveyor);
	                END_REGION

	                REGION MCO

	                    #sFB_MCOConveyLinxAixController550(iUDT_AixConfig := #iUDT_Configuration."550".MCO_M01,
	                                                       iUDT_AixInputsModule := #iUDT_MotorInput550,
	                                                       ix_24vOk := #ix_24vOk,
	                                                       ix_SimulationModeActive := "DB_Memory".Simulation,
	                                                       ii_MotorPositionId := 1,
	                                                       qUDT_HMIStatus => #iqUDT_WorkstationStatus."550".MCO_M01,
	                                                       iqUDT_AixOutputsModule := #iqUDT_MotorOutput550,
	                                                       iqUDT_ConveyorInterface := #sUDT_Interface550,
	                                                       iqUDT_MCOStatistics := #iqUDT_WorkstationStatistics."550".MCO_M01);
	                END_REGION
	            END_REGION

	            REGION 560

	                REGION Displacement

	                    #sFB_Displacement560(#sUDT_Interface560);

	                END_REGION

	                REGION Tracking

	                    #sFB_Tracking560(iUDT_ConveyorCommonConfiguration := #iUDT_Configuration."560".Conveyor.Common,
	                                     iqa_TrackingData := #sa_TrackingArray560,
	                                     iqUDT_ConveyorInterface := #sUDT_Interface560,
	                                     iqUDT_HandshakeUp := #sUDT_Handshake550,
	                                     iqUDT_Handshake := #sUDT_Handshake560);
	                END_REGION

	                REGION EOS

	                    #sFB_PECUpdate560(iUDT_PECUpdateConfiguration := #iUDT_Configuration."560".PEC_Eos,
	                                      iUDT_ConveyorCommonConfiguration := #iUDT_Configuration."560".Conveyor.Common,
	                                      ix_PEC := NOT #iUDT_MotorInput550.AllSensorPortInputs.RightSensor,
	                                      ix_TeachingMode := FALSE,
	                                      qUDT_Status => #iqUDT_WorkstationStatus."560".PEC_EoS,
	                                      qi_GINwrite => #ti_dummy,
	                                      qx_PECFiltered => #tx_dummy,
	                                      iqa_TrackingData := #sa_TrackingArray560,
	                                      iqUDT_ConveyorInterface := #sUDT_Interface560,
	                                      iqUDT_UnknownGINRange := #iqUDT_UnknownGINRange,
	                                      iqUDT_FifoHeader := "DB_FIFOLostGIN".Header,
	                                      iqa_FifoData := "DB_FIFOLostGIN".Data,
	                                      iqUDT_Statistics := #iqUDT_WorkstationStatistics."560".PEC_EoS);

	                END_REGION

	                REGION Conveyor

	                    #sUDT_Handshake560.RTR := #sx_RightIndexing AND
	                    ((#iqUDT_WorkstationStatus."570".PEC_EoS.PEC AND #sUDT_Interface570.ActualSpeed <> 0) OR #iqUDT_WorkstationStatus."560".PEC_EoS.PEC);

	                    #sFB_Conveyor560(iUDT_ConveyorConfiguration := #iUDT_Configuration."560".Conveyor,
	                                     idi_PECEoSDistance := #iUDT_Configuration."560".PEC_Eos.Distance,
	                                     idi_PECBoSDistance := 0,
	                                     ii_ExternalSpeed := 0,
	                                     ix_SafetyOk := #ix_SafetyOk,
	                                     ix_24vOk := #ix_24vOk,
	                                     ix_400vOk := #ix_400vOk,
	                                     ix_HardwareOk := #ix_HardwareOk,
	                                     ix_PECEoS := #iqUDT_WorkstationStatus."560".PEC_EoS.PEC,
	                                     ix_PECBoS := TRUE,
	                                     ix_ReverseDirection := FALSE,
	                                     ix_ExternalRequestDieBack := FALSE,
	                                     ix_ExternalRequestHold := #sx_RightExternalRequestHold560,
	                                     ix_ResetEnergySave := FALSE,
	                                     qUDT_HMIStatus => #iqUDT_WorkstationStatus."560".Conveyor,
	                                     qUDT_Status => #iqUDT_WorkstationCommonStatus."560",
	                                     iqUDT_EquipmentControl := #iqUDT_EquipmentControl,
	                                     iqUDT_ConveyorCommand := #iqUDT_WorkstationCommands."560".Conveyor,
	                                     iqUDT_ConveyorInterface := #sUDT_Interface560,
	                                     iqUDT_HandShakeUp := #sUDT_Handshake550,
	                                     iqUDT_HandShake := #sUDT_Handshake560,
	                                     iqUDT_Statistics := #iqUDT_WorkstationStatistics."560".Conveyor);
	                END_REGION

	                REGION MCO

	                    #sFB_MCOConveyLinxAixController560(iUDT_AixConfig := #iUDT_Configuration."560".MCO_M01,
	                                                       iUDT_AixInputsModule := #iUDT_MotorInput550,
	                                                       ix_24vOk := #ix_24vOk,
	                                                       ix_SimulationModeActive := "DB_Memory".Simulation,
	                                                       ii_MotorPositionId := 2,
	                                                       qUDT_HMIStatus => #iqUDT_WorkstationStatus."560".MCO_M01,
	                                                       iqUDT_AixOutputsModule := #iqUDT_MotorOutput550,
	                                                       iqUDT_ConveyorInterface := #sUDT_Interface560,
	                                                       iqUDT_MCOStatistics := #iqUDT_WorkstationStatistics."560".MCO_M01);
	                END_REGION

	            END_REGION

	            REGION 570

	                REGION Displacement

	                    #sFB_Displacement570(#sUDT_Interface570);

	                END_REGION

	                REGION Tracking

	                    #sFB_Tracking570(iUDT_ConveyorCommonConfiguration := #iUDT_Configuration."570".Conveyor.Common,
	                                     iqa_TrackingData := #sa_TrackingArray570,
	                                     iqUDT_ConveyorInterface := #sUDT_Interface570,
	                                     iqUDT_HandshakeUp := #sUDT_Handshake560,
	                                     iqUDT_Handshake := #sUDT_Handshake570);
	                END_REGION

	                REGION EOS

	                    #sFB_PECUpdate570(iUDT_PECUpdateConfiguration := #iUDT_Configuration."570".PEC_Eos,
	                                      iUDT_ConveyorCommonConfiguration := #iUDT_Configuration."570".Conveyor.Common,
	                                      ix_PEC := NOT #iUDT_MotorInput570.AllSensorPortInputs.LeftSensor,
	                                      ix_TeachingMode := FALSE,
	                                      qUDT_Status => #iqUDT_WorkstationStatus."570".PEC_EoS,
	                                      qi_GINwrite => #ti_dummy,
	                                      qx_PECFiltered => #tx_dummy,
	                                      iqa_TrackingData := #sa_TrackingArray570,
	                                      iqUDT_ConveyorInterface := #sUDT_Interface570,
	                                      iqUDT_UnknownGINRange := #iqUDT_UnknownGINRange,
	                                      iqUDT_FifoHeader := "DB_FIFOLostGIN".Header,
	                                      iqa_FifoData := "DB_FIFOLostGIN".Data,
	                                      iqUDT_Statistics := #iqUDT_WorkstationStatistics."570".PEC_EoS);

	                END_REGION

	                REGION Conveyor

	                    #sUDT_Handshake570.RTR := #sx_RightIndexing AND
	                    ((#iqUDT_WorkstationStatus."580".PEC_EoS.PEC AND #sUDT_Interface580.ActualSpeed <> 0) OR #iqUDT_WorkstationStatus."570".PEC_EoS.PEC);

	                    #sFB_Conveyor570(iUDT_ConveyorConfiguration := #iUDT_Configuration."570".Conveyor,
	                                     idi_PECEoSDistance := #iUDT_Configuration."570".PEC_Eos.Distance,
	                                     idi_PECBoSDistance := 0,
	                                     ii_ExternalSpeed := 0,
	                                     ix_SafetyOk := #ix_SafetyOk,
	                                     ix_24vOk := #ix_24vOk,
	                                     ix_400vOk := #ix_400vOk,
	                                     ix_HardwareOk := #ix_HardwareOk,
	                                     ix_PECEoS := #iqUDT_WorkstationStatus."570".PEC_EoS.PEC,
	                                     ix_PECBoS := TRUE,
	                                     ix_ExternalRequestHold := #sx_RightExternalRequestHold570,
	                                     qUDT_HMIStatus => #iqUDT_WorkstationStatus."570".Conveyor,
	                                     qUDT_Status => #iqUDT_WorkstationCommonStatus."570",
	                                     iqUDT_EquipmentControl := #iqUDT_EquipmentControl,
	                                     iqUDT_ConveyorCommand := #iqUDT_WorkstationCommands."570".Conveyor,
	                                     iqUDT_ConveyorInterface := #sUDT_Interface570,
	                                     iqUDT_HandShakeUp := #sUDT_Handshake560,
	                                     iqUDT_HandShake := #sUDT_Handshake570,
	                                     iqUDT_Statistics := #iqUDT_WorkstationStatistics."570".Conveyor);
	                END_REGION

	                REGION MCO

	                    #sFB_MCOConveyLinxAixController570(iUDT_AixConfig := #iUDT_Configuration."570".MCO_M01,
	                                                       iUDT_AixInputsModule := #iUDT_MotorInput570,
	                                                       ix_24vOk := #ix_24vOk,
	                                                       ix_SimulationModeActive := "DB_Memory".Simulation,
	                                                       ii_MotorPositionId := 1,
	                                                       qUDT_HMIStatus => #iqUDT_WorkstationStatus."570".MCO_M01,
	                                                       iqUDT_AixOutputsModule := #iqUDT_MotorOutput570,
	                                                       iqUDT_ConveyorInterface := #sUDT_Interface570,
	                                                       iqUDT_MCOStatistics := #iqUDT_WorkstationStatistics."570".MCO_M01);
	                END_REGION
	            END_REGION

	            REGION 580

	                REGION Displacement

	                    #sFB_Displacement580(#sUDT_Interface580);

	                END_REGION

	                REGION Tracking

	                    #sFB_Tracking580(iUDT_ConveyorCommonConfiguration := #iUDT_Configuration."580".Conveyor.Common,
	                                     iqa_TrackingData := #sa_TrackingArray580,
	                                     iqUDT_ConveyorInterface := #sUDT_Interface580,
	                                     iqUDT_HandshakeUp := #sUDT_Handshake570,
	                                     iqUDT_Handshake := #sUDT_Handshake580);
	                END_REGION

	                REGION EOS

	                    #sFB_PECUpdate580(iUDT_PECUpdateConfiguration := #iUDT_Configuration."580".PEC_Eos,
	                                      iUDT_ConveyorCommonConfiguration := #iUDT_Configuration."580".Conveyor.Common,
	                                      ix_PEC := NOT #iUDT_MotorInput570.AllSensorPortInputs.RightSensor,
	                                      ix_TeachingMode := FALSE,
	                                      qUDT_Status => #iqUDT_WorkstationStatus."580".PEC_EoS,
	                                      qi_GINwrite => #ti_dummy,
	                                      qx_PECFiltered => #tx_dummy,
	                                      iqa_TrackingData := #sa_TrackingArray580,
	                                      iqUDT_ConveyorInterface := #sUDT_Interface580,
	                                      iqUDT_UnknownGINRange := #iqUDT_UnknownGINRange,
	                                      iqUDT_FifoHeader := "DB_FIFOLostGIN".Header,
	                                      iqa_FifoData := "DB_FIFOLostGIN".Data,
	                                      iqUDT_Statistics := #iqUDT_WorkstationStatistics."580".PEC_EoS);

	                END_REGION

	                REGION Conveyor

	                    #sUDT_Handshake580.RTR := #sx_RightIndexing AND
	                    ((#iqUDT_WorkstationStatus."590".PEC_EoS.PEC AND #sUDT_Interface590.ActualSpeed <> 0) OR #iqUDT_WorkstationStatus."580".PEC_EoS.PEC);

	                    #sFB_Conveyor580(iUDT_ConveyorConfiguration := #iUDT_Configuration."580".Conveyor,
	                                     idi_PECEoSDistance := #iUDT_Configuration."580".PEC_Eos.Distance,
	                                     idi_PECBoSDistance := 0,
	                                     ii_ExternalSpeed := 0,
	                                     ix_SafetyOk := #ix_SafetyOk,
	                                     ix_24vOk := #ix_24vOk,
	                                     ix_400vOk := #ix_400vOk,
	                                     ix_HardwareOk := #ix_HardwareOk,
	                                     ix_PECEoS := #iqUDT_WorkstationStatus."580".PEC_EoS.PEC,
	                                     ix_PECBoS := TRUE,
	                                     ix_ReverseDirection := FALSE,
	                                     ix_ExternalRequestDieBack := FALSE,
	                                     ix_ExternalRequestHold := #sx_RightExternalRequestHold580,
	                                     ix_ResetEnergySave := FALSE,
	                                     qUDT_HMIStatus => #iqUDT_WorkstationStatus."580".Conveyor,
	                                     qUDT_Status => #iqUDT_WorkstationCommonStatus."580",
	                                     iqUDT_EquipmentControl := #iqUDT_EquipmentControl,
	                                     iqUDT_ConveyorCommand := #iqUDT_WorkstationCommands."580".Conveyor,
	                                     iqUDT_ConveyorInterface := #sUDT_Interface580,
	                                     iqUDT_HandShakeUp := #sUDT_Handshake570,
	                                     iqUDT_HandShake := #sUDT_Handshake580,
	                                     iqUDT_Statistics := #iqUDT_WorkstationStatistics."580".Conveyor);
	                END_REGION

	                REGION MCO

	                    #sFB_MCOConveyLinxAixController580(iUDT_AixConfig := #iUDT_Configuration."580".MCO_M01,
	                                                       iUDT_AixInputsModule := #iUDT_MotorInput570,
	                                                       ix_24vOk := #ix_24vOk,
	                                                       ix_SimulationModeActive := "DB_Memory".Simulation,
	                                                       ii_MotorPositionId := 2,
	                                                       qUDT_HMIStatus => #iqUDT_WorkstationStatus."580".MCO_M01,
	                                                       iqUDT_AixOutputsModule := #iqUDT_MotorOutput570,
	                                                       iqUDT_ConveyorInterface := #sUDT_Interface580,
	                                                       iqUDT_MCOStatistics := #iqUDT_WorkstationStatistics."580".MCO_M01);
	                END_REGION

	            END_REGION

	            REGION 590

	                REGION Displacement

	                    #sFB_Displacement590(#sUDT_Interface590);

	                END_REGION

	                REGION Tracking

	                    #sFB_Tracking590(iUDT_ConveyorCommonConfiguration := #iUDT_Configuration."590".Conveyor.Common,
	                                     iqa_TrackingData := #sa_TrackingArray590,
	                                     iqUDT_ConveyorInterface := #sUDT_Interface590,
	                                     iqUDT_HandshakeUp := #sUDT_Handshake580,
	                                     iqUDT_Handshake := #sUDT_Handshake590);
	                END_REGION

	                REGION EOS

	                    #sFB_PECUpdate590(iUDT_PECUpdateConfiguration := #iUDT_Configuration."590".PEC_Eos,
	                                      iUDT_ConveyorCommonConfiguration := #iUDT_Configuration."590".Conveyor.Common,
	                                      ix_PEC := NOT #iUDT_MotorInput590.AllSensorPortInputs.LeftSensor,
	                                      ix_TeachingMode := FALSE,
	                                      qUDT_Status => #iqUDT_WorkstationStatus."590".PEC_EoS,
	                                      qi_GINwrite => #ti_dummy,
	                                      qx_PECFiltered => #tx_dummy,
	                                      iqa_TrackingData := #sa_TrackingArray590,
	                                      iqUDT_ConveyorInterface := #sUDT_Interface590,
	                                      iqUDT_UnknownGINRange := #iqUDT_UnknownGINRange,
	                                      iqUDT_FifoHeader := "DB_FIFOLostGIN".Header,
	                                      iqa_FifoData := "DB_FIFOLostGIN".Data,
	                                      iqUDT_Statistics := #iqUDT_WorkstationStatistics."590".PEC_EoS);

	                END_REGION

	                REGION Conveyor

	                    #sUDT_Handshake590.RTR := (#sx_RightIndexing AND #iqUDT_WorkstationStatus."590".PEC_EoS.PEC)
	                    OR (#sx_RightPushOutActiveStation1 AND #iqUDT_WorkstationStatus."610".PEC_EoS.PEC AND #sUDT_Interface611.ActualSpeed <> 0);

	                    #sFB_Conveyor590(iUDT_ConveyorConfiguration := #iUDT_Configuration."590".Conveyor,
	                                     idi_PECEoSDistance := #iUDT_Configuration."590".PEC_Eos.Distance,
	                                     idi_PECBoSDistance := 0,
	                                     ii_ExternalSpeed := 0,
	                                     ix_SafetyOk := #ix_SafetyOk,
	                                     ix_24vOk := #ix_24vOk,
	                                     ix_400vOk := #ix_400vOk,
	                                     ix_HardwareOk := #ix_HardwareOk,
	                                     ix_PECEoS := #iqUDT_WorkstationStatus."590".PEC_EoS.PEC,
	                                     ix_PECBoS := TRUE,
	                                     ix_ReverseDirection := FALSE,
	                                     ix_ExternalRequestDieBack := FALSE,
	                                     ix_ExternalRequestHold := #sx_RightExternalRequestHold590,
	                                     ix_ResetEnergySave := FALSE,
	                                     qUDT_HMIStatus => #iqUDT_WorkstationStatus."590".Conveyor,
	                                     qUDT_Status => #iqUDT_WorkstationCommonStatus."590",
	                                     iqUDT_EquipmentControl := #iqUDT_EquipmentControl,
	                                     iqUDT_ConveyorCommand := #iqUDT_WorkstationCommands."590".Conveyor,
	                                     iqUDT_ConveyorInterface := #sUDT_Interface590,
	                                     iqUDT_HandShakeUp := #sUDT_Handshake580,
	                                     iqUDT_HandShake := #sUDT_Handshake590,
	                                     iqUDT_Statistics := #iqUDT_WorkstationStatistics."590".Conveyor);
	                END_REGION

	                REGION MCO

	                    #sFB_MCOConveyLinxAixController590(iUDT_AixConfig := #iUDT_Configuration."590".MCO_M01,
	                                                       iUDT_AixInputsModule := #iUDT_MotorInput590,
	                                                       ix_24vOk := #ix_24vOk,
	                                                       ix_SimulationModeActive := "DB_Memory".Simulation,
	                                                       ii_MotorPositionId := 1,
	                                                       qUDT_HMIStatus => #iqUDT_WorkstationStatus."590".MCO_M01,
	                                                       iqUDT_AixOutputsModule := #iqUDT_MotorOutput590,
	                                                       iqUDT_ConveyorInterface := #sUDT_Interface590,
	                                                       iqUDT_MCOStatistics := #iqUDT_WorkstationStatistics."590".MCO_M01);
	                END_REGION
	            END_REGION

	            REGION 610

	                REGION Displacement

	                    #sFB_Displacement610(#sUDT_Interface610);

	                END_REGION

	                REGION MCO

	                    #sFB_MCOConveyLinxAixController610(iUDT_AixConfig := #iUDT_Configuration."610".MCO_M01,
	                                                       iUDT_AixInputsModule := #iUDT_MotorInput610,
	                                                       ix_24vOk := #ix_24vOk,
	                                                       ix_SimulationModeActive := "DB_Memory".Simulation,
	                                                       ii_MotorPositionId := 1,
	                                                       qUDT_HMIStatus => #iqUDT_WorkstationStatus."610".MCO_M01,
	                                                       iqUDT_AixOutputsModule := #iqUDT_MotorOutput610,
	                                                       iqUDT_ConveyorInterface := #sUDT_Interface610,
	                                                       iqUDT_MCOStatistics := #iqUDT_WorkstationStatistics."610".MCO_M01);
	                END_REGION
	            END_REGION

	            REGION 611

	                REGION Displacement

	                    #sFB_Displacement611(#sUDT_Interface611);

	                END_REGION

	                REGION RAT

	                    #sFB_RightAngledTransfer611(iUDT_Configuration := #iUDT_Configuration."611".RightAngledTransfer,
	                                                iUDT_LowerConveyorConfiguration := #iUDT_Configuration."610".Conveyor,
	                                                iUDT_UpperConveyorConfiguration := #iUDT_Configuration."611".Conveyor,
	                                                iUDT_PECConfiguration := #iUDT_Configuration."610".PEC_EoS,
	                                                ii_DestinationA := 0,
	                                                ii_DestinationB := 0,
	                                                ii_DestinationC := 0,
	                                                ii_DestinationD := 1,
	                                                ix_HardwareOk := #ix_HardwareOk,
	                                                ix_400vOk := #ix_400vOk,
	                                                ix_24vOk := #ix_24vOk,
	                                                ix_SafetyOk := #ix_SafetyOk,
	                                                ix_AirPressureOk := #ix_AirPressureOk,
	                                                ix_SectionIsDown := #ix_SectionIsDown611,
	                                                ix_SectionIsUp := #ix_SectionIsUp611,
	                                                ix_ConveyorAAuto := false,
	                                                ix_ConveyorBAuto := false,
	                                                ix_ConveyorCAuto := FALSE,
	                                                ix_ConveyorDAuto := #iqUDT_WorkstationCommonStatus."590".AutoON,
	                                                ix_PEC := #iUDT_MotorInput610.AllSensorPortInputs.LeftSensor,
	                                                ix_ExternalReceiveRequestA := FALSE,
	                                                ix_ExternalReceiveRequestB := FALSE,
	                                                ix_ExternalReceiveRequestC := FALSE,
	                                                ix_ExternalReceiveRequestD := #sx_RightPushOutActiveStation1,
	                                                ix_PECInfeedD := #iqUDT_WorkstationStatus."590".PEC_EoS.PEC,
	                                                qUDT_HMIRATStatus => #iqUDT_WorkstationStatus."611".RightAngledTransfer,
	                                                qUDT_HMIConveyorStatus => #iqUDT_WorkstationStatus."610".Conveyor,
	                                                qUDT_HMIPECStatus => #iqUDT_WorkstationStatus."610".PEC_EoS,
	                                                qUDT_RATStatus => #iqUDT_WorkstationCommonStatus."611",
	                                                qUDT_ConveyorStatus => #iqUDT_WorkstationCommonStatus."610",
	                                                qx_PopupControl => #qx_PopupControl611,
	                                                qx_ExternalSendRequestA => #tx_dummy,
	                                                qx_ExternalSendRequestB => #tx_dummy,
	                                                qx_ExternalSendRequestC => #tx_dummy,
	                                                qx_ExternalSendRequestD => #tx_dummy,
	                                                iqUDT_EquipmentControl := #iqUDT_EquipmentControl,
	                                                iqUDT_RATCommand := #iqUDT_WorkstationCommands."611".RightAngledTransfer,
	                                                iqUDT_ConveyorCommand := #iqUDT_WorkstationCommands."610".Conveyor,
	                                                iqUDT_RATStatistics := #iqUDT_WorkstationStatistics."611".RightAngledTransfer,
	                                                iqUDT_ConveyorStatistics := #iqUDT_WorkstationStatistics."610".Conveyor,
	                                                iqUDT_PECStatistics := #iqUDT_WorkstationStatistics."610".PEC_EoS,
	                                                iqUDT_HandShakeConveyorA := #tUDT_DummyConveyorHandshake,
	                                                iqUDT_HandShakeConveyorB := #sUDT_Handshake610,
	                                                iqUDT_HandShakeConveyorC := #sUDT_Handshake590,
	                                                iqUDT_HandShakeConveyorD := #tUDT_DummyConveyorHandshake,
	                                                iqUDT_LowerConveyorInterface := #sUDT_Interface610,
	                                                iqUDT_UpperConveyorInterface := #sUDT_Interface611,
	                                                iqUDT_RATPositioning := #iqUDT_RATPositioning610,
	                                                iqUDT_BladeStopEoSInterface := #tUDT_DummyBladeStop,
	                                                iqUDT_BladeStopBoSInterface := #tUDT_DummyBladeStop);

	                END_REGION

	                REGION MCO

	                    #sFB_MCOConveyLinxAixController611(iUDT_AixConfig := #iUDT_Configuration."611".MCO_M01,
	                                                       iUDT_AixInputsModule := #iUDT_MotorInput610,
	                                                       ii_PositionSetpoint := #iqUDT_RATPositioning610.Upper.EndPosition,
	                                                       ix_24vOk := #ix_24vOk,
	                                                       ix_SimulationModeActive := "DB_Memory".Simulation,
	                                                       ii_MotorPositionId := 2,
	                                                       ix_StartPositioning := #iqUDT_RATPositioning610.Upper.Start,
	                                                       ix_ResetPosition := #iqUDT_RATPositioning610.Upper.ResetPosition,
	                                                       qUDT_HMIStatus => #iqUDT_WorkstationStatus."611".MCO_M01,
	                                                       qx_Positioned => #iqUDT_RATPositioning610.Upper.Done,
	                                                       iqUDT_AixOutputsModule := #iqUDT_MotorOutput610,
	                                                       iqUDT_ConveyorInterface := #sUDT_Interface611,
	                                                       iqUDT_MCOStatistics := #iqUDT_WorkstationStatistics."611".MCO_M01);
	                END_REGION

	            END_REGION

	            REGION 620

	                REGION Displacement

	                    #sFB_Displacement620(#sUDT_Interface620);

	                END_REGION

	                REGION MCO

	                    #sFB_MCOConveyLinxAixController620(iUDT_AixConfig := #iUDT_Configuration."620".MCO_M01,
	                                                       iUDT_AixInputsModule := #iUDT_MotorInput620,
	                                                       ii_PositionSetpoint := #iqUDT_RATPositioning620.Lower.EndPosition,
	                                                       ix_24vOk := #ix_24vOk,
	                                                       ix_SimulationModeActive := "DB_Memory".Simulation,
	                                                       ii_MotorPositionId := 1,
	                                                       ix_StartPositioning := #iqUDT_RATPositioning620.Lower.Start,
	                                                       ix_ResetPosition := #iqUDT_RATPositioning620.Lower.ResetPosition,
	                                                       qUDT_HMIStatus => #iqUDT_WorkstationStatus."620".MCO_M01,
	                                                       qx_Positioned => #iqUDT_RATPositioning620.Lower.Done,
	                                                       iqUDT_AixOutputsModule := #iqUDT_MotorOutput620,
	                                                       iqUDT_ConveyorInterface := #sUDT_Interface620,
	                                                       iqUDT_MCOStatistics := #iqUDT_WorkstationStatistics."620".MCO_M01);
	                END_REGION
	            END_REGION

	            REGION 621

	                REGION Displacement

	                    #sFB_Displacement621(#sUDT_Interface621);

	                END_REGION

	                REGION RAT

	                    #sFB_RightAngledTransfer621(iUDT_Configuration := #iUDT_Configuration."621".RightAngledTransfer,
	                                                iUDT_LowerConveyorConfiguration := #iUDT_Configuration."620".Conveyor,
	                                                iUDT_UpperConveyorConfiguration := #iUDT_Configuration."621".Conveyor,
	                                                iUDT_PECConfiguration := #iUDT_Configuration."620".PEC_EoS,
	                                                ii_DestinationA := 1,
	                                                ii_DestinationB := 0,
	                                                ii_DestinationC := 0,
	                                                ii_DestinationD := 1,
	                                                ix_HardwareOk := #ix_HardwareOk,
	                                                ix_400vOk := #ix_400vOk,
	                                                ix_24vOk := #ix_24vOk,
	                                                ix_SafetyOk := #ix_SafetyOk,
	                                                ix_AirPressureOk := #ix_AirPressureOk,
	                                                ix_SectionIsDown := #ix_SectionIsDown621,
	                                                ix_SectionIsUp := #ix_SectionIsUp621,
	                                                ix_ConveyorAAuto := #iqUDT_WorkstationCommonStatus."610".AutoON,
	                                                ix_ConveyorBAuto := false,
	                                                ix_ConveyorCAuto := false,
	                                                ix_ConveyorDAuto := #iqUDT_WorkstationCommonStatus."750".AutoON,
	                                                ix_PEC := #iUDT_MotorInput620.AllSensorPortInputs.LeftSensor,
	                                                ix_ExternalReceiveRequestA := NOT #iqUDT_WorkstationStatus."610".PEC_EoS.PEC,
	                                                ix_ExternalReceiveRequestB := FALSE,
	                                                ix_ExternalReceiveRequestC := FALSE,
	                                                ix_ExternalReceiveRequestD := NOT #iqUDT_WorkstationStatus."750".PEC_EoS.PEC,
	                                                ix_PECInfeedA := #iqUDT_WorkstationStatus."610".PEC_EoS.PEC,
	                                                ix_PECInfeedD := #iqUDT_WorkstationStatus."750".PEC_EoS.PEC,
	                                                qUDT_HMIRATStatus => #iqUDT_WorkstationStatus."621".RightAngledTransfer,
	                                                qUDT_HMIConveyorStatus => #iqUDT_WorkstationStatus."620".Conveyor,
	                                                qUDT_HMIPECStatus => #iqUDT_WorkstationStatus."620".PEC_EoS,
	                                                qUDT_RATStatus => #iqUDT_WorkstationCommonStatus."621",
	                                                qUDT_ConveyorStatus => #iqUDT_WorkstationCommonStatus."620",
	                                                qx_PopupControl => #qx_PopupControl621,
	                                                qx_ExternalSendRequestA => #tx_dummy,
	                                                qx_ExternalSendRequestB => #tx_dummy,
	                                                qx_ExternalSendRequestC => #tx_dummy,
	                                                qx_ExternalSendRequestD => #tx_dummy,
	                                                iqUDT_EquipmentControl := #iqUDT_EquipmentControl,
	                                                iqUDT_RATCommand := #iqUDT_WorkstationCommands."621".RightAngledTransfer,
	                                                iqUDT_ConveyorCommand := #iqUDT_WorkstationCommands."620".Conveyor,
	                                                iqUDT_RATStatistics := #iqUDT_WorkstationStatistics."621".RightAngledTransfer,
	                                                iqUDT_ConveyorStatistics := #iqUDT_WorkstationStatistics."620".Conveyor,
	                                                iqUDT_PECStatistics := #iqUDT_WorkstationStatistics."620".PEC_EoS,
	                                                iqUDT_HandShakeConveyorA := #sUDT_Handshake610,
	                                                iqUDT_HandShakeConveyorB := #sUDT_Handshake620,
	                                                iqUDT_HandShakeConveyorC := #tUDT_DummyConveyorHandshake,
	                                                iqUDT_HandShakeConveyorD := #sUDT_Handshake750,
	                                                iqUDT_LowerConveyorInterface := #sUDT_Interface620,
	                                                iqUDT_UpperConveyorInterface := #sUDT_Interface621,
	                                                iqUDT_RATPositioning := #iqUDT_RATPositioning620,
	                                                iqUDT_BladeStopEoSInterface := #tUDT_DummyBladeStop,
	                                                iqUDT_BladeStopBoSInterface := #tUDT_DummyBladeStop);

	                END_REGION

	                REGION MCO

	                    #sFB_MCOConveyLinxAixController621(iUDT_AixConfig := #iUDT_Configuration."621".MCO_M01,
	                                                       iUDT_AixInputsModule := #iUDT_MotorInput620,
	                                                       ii_PositionSetpoint := #iqUDT_RATPositioning620.Upper.EndPosition,
	                                                       ix_24vOk := #ix_24vOk,
	                                                       ix_SimulationModeActive := "DB_Memory".Simulation,
	                                                       ii_MotorPositionId := 2,
	                                                       ix_StartPositioning := #iqUDT_RATPositioning620.Upper.Start,
	                                                       ix_ResetPosition := #iqUDT_RATPositioning620.Upper.ResetPosition,
	                                                       qUDT_HMIStatus => #iqUDT_WorkstationStatus."621".MCO_M01,
	                                                       qx_Positioned => #iqUDT_RATPositioning620.Upper.Done,
	                                                       iqUDT_AixOutputsModule := #iqUDT_MotorOutput620,
	                                                       iqUDT_ConveyorInterface := #sUDT_Interface621,
	                                                       iqUDT_MCOStatistics := #iqUDT_WorkstationStatistics."621".MCO_M01);
	                END_REGION

	            END_REGION

	            REGION 630

	                REGION Displacement

	                    #sFB_Displacement630(#sUDT_Interface630);

	                END_REGION

	                REGION Conveyor

	                    #sFB_Conveyor630(iUDT_ConveyorConfiguration := #iUDT_Configuration."630".Conveyor,
	                                     idi_PECEoSDistance := 0,
	                                     idi_PECBoSDistance := 0,
	                                     ii_ExternalSpeed := 0,
	                                     ix_SafetyOk := #ix_SafetyOk,
	                                     ix_24vOk := #ix_24vOk,
	                                     ix_400vOk := #ix_400vOk,
	                                     ix_HardwareOk := #ix_HardwareOk,
	                                     ix_PECEoS := TRUE,
	                                     ix_PECBoS := TRUE,
	                                     ix_ReverseDirection := FALSE,
	                                     ix_ExternalRequestDieBack := FALSE,
	                                     ix_ExternalRequestHold := FALSE,
	                                     ix_ResetEnergySave := FALSE,
	                                     qUDT_HMIStatus => #iqUDT_WorkstationStatus."630".Conveyor,
	                                     qUDT_Status => #iqUDT_WorkstationCommonStatus."630",
	                                     iqUDT_EquipmentControl := #iqUDT_EquipmentControl,
	                                     iqUDT_ConveyorCommand := #iqUDT_WorkstationCommands."630".Conveyor,
	                                     iqUDT_ConveyorInterface := #sUDT_Interface630,
	                                     iqUDT_HandShakeUp := #sUDT_Handshake620,
	                                     iqUDT_HandShake := #iqUDT_HandshakeDownstream630,
	                                     iqUDT_Statistics := #iqUDT_WorkstationStatistics."630".Conveyor);
	                END_REGION

	                REGION MCO

	                    #sFB_MCOConveyLinxAixController630(iUDT_AixConfig := #iUDT_Configuration."630".MCO_M01,
	                                                       iUDT_AixInputsModule := #iUDT_MotorInput630,
	                                                       ix_24vOk := #ix_24vOk,
	                                                       ix_SimulationModeActive := "DB_Memory".Simulation,
	                                                       ii_MotorPositionId := 1,
	                                                       qUDT_HMIStatus => #iqUDT_WorkstationStatus."630".MCO_M01,
	                                                       iqUDT_AixOutputsModule := #iqUDT_MotorOutput630,
	                                                       iqUDT_ConveyorInterface := #sUDT_Interface630,
	                                                       iqUDT_MCOStatistics := #iqUDT_WorkstationStatistics."630".MCO_M01);
	                END_REGION
	            END_REGION

	            REGION 710

	                REGION Displacement

	                    #sFB_Displacement710(#sUDT_Interface710);

	                END_REGION

	                REGION EOS
	                    #sFB_PEC710(ix_PEC := NOT #iUDT_MotorInput710.AllSensorPortInputs.LeftSensor,
	                                iUDT_PECConfiguration := #iUDT_Configuration."710".PEC_Eos,
	                                qx_PECFiltered => #tx_dummy,
	                                qUDT_HMIStatus => #iqUDT_WorkstationStatus."710".PEC_EoS,
	                                iqUDT_ConveyorInterface := #sUDT_Interface710,
	                                iqUDT_PECStatistics := #iqUDT_WorkstationStatistics."710".PEC_EoS);

	                END_REGION

	                REGION Conveyor

	                    #sFB_Conveyor710(iUDT_ConveyorConfiguration := #iUDT_Configuration."710".Conveyor,
	                                     idi_PECEoSDistance := #iUDT_Configuration."710".PEC_Eos.Distance,
	                                     idi_PECBoSDistance := 0,
	                                     ii_ExternalSpeed := 0,
	                                     ix_SafetyOk := #ix_SafetyOk,
	                                     ix_24vOk := #ix_24vOk,
	                                     ix_400vOk := #ix_400vOk,
	                                     ix_HardwareOk := #ix_HardwareOk,
	                                     ix_PECEoS := #iqUDT_WorkstationStatus."710".PEC_EoS.PEC,
	                                     ix_PECBoS := TRUE,
	                                     ix_ReverseDirection := FALSE,
	                                     ix_ExternalRequestDieBack := FALSE,
	                                     ix_ExternalRequestHold := #sx_RightExternalRequestHold710,
	                                     ix_ResetEnergySave := FALSE,
	                                     qUDT_HMIStatus => #iqUDT_WorkstationStatus."710".Conveyor,
	                                     qUDT_Status => #iqUDT_WorkstationCommonStatus."710",
	                                     iqUDT_EquipmentControl := #iqUDT_EquipmentControl,
	                                     iqUDT_ConveyorCommand := #iqUDT_WorkstationCommands."710".Conveyor,
	                                     iqUDT_ConveyorInterface := #sUDT_Interface710,
	                                     iqUDT_HandShakeUp := #tUDT_DummyConveyorHandshake,
	                                     iqUDT_HandShake := #sUDT_Handshake710,
	                                     iqUDT_Statistics := #iqUDT_WorkstationStatistics."710".Conveyor);
	                END_REGION

	                REGION MCO

	                    #sFB_MCOConveyLinxAixController710(iUDT_AixConfig := #iUDT_Configuration."710".MCO_M01,
	                                                       iUDT_AixInputsModule := #iUDT_MotorInput710,
	                                                       ix_24vOk := #ix_24vOk,
	                                                       ix_SimulationModeActive := "DB_Memory".Simulation,
	                                                       ii_MotorPositionId := 1,
	                                                       qUDT_HMIStatus => #iqUDT_WorkstationStatus."710".MCO_M01,
	                                                       iqUDT_AixOutputsModule := #iqUDT_MotorOutput710,
	                                                       iqUDT_ConveyorInterface := #sUDT_Interface710,
	                                                       iqUDT_MCOStatistics := #iqUDT_WorkstationStatistics."710".MCO_M01);
	                END_REGION

	            END_REGION

	            REGION 720

	                REGION Displacement

	                    #sFB_Displacement720(#sUDT_Interface720);

	                END_REGION

	                REGION EOS
	                    #sFB_PEC720(ix_PEC := NOT #iUDT_MotorInput710.AllSensorPortInputs.RightSensor,
	                                iUDT_PECConfiguration := #iUDT_Configuration."720".PEC_Eos,
	                                qx_PECFiltered => #tx_dummy,
	                                qUDT_HMIStatus => #iqUDT_WorkstationStatus."720".PEC_EoS,
	                                iqUDT_ConveyorInterface := #sUDT_Interface720,
	                                iqUDT_PECStatistics := #iqUDT_WorkstationStatistics."720".PEC_EoS);


	                END_REGION

	                REGION Conveyor

	                    #sFB_Conveyor720(iUDT_ConveyorConfiguration := #iUDT_Configuration."720".Conveyor,
	                                     idi_PECEoSDistance := #iUDT_Configuration."720".PEC_Eos.Distance,
	                                     idi_PECBoSDistance := 0,
	                                     ii_ExternalSpeed := 0,
	                                     ix_SafetyOk := #ix_SafetyOk,
	                                     ix_24vOk := #ix_24vOk,
	                                     ix_400vOk := #ix_400vOk,
	                                     ix_HardwareOk := #ix_HardwareOk,
	                                     ix_PECEoS := #iqUDT_WorkstationStatus."720".PEC_EoS.PEC,
	                                     ix_PECBoS := TRUE,
	                                     ix_ReverseDirection := FALSE,
	                                     ix_ExternalRequestDieBack := FALSE,
	                                     ix_ExternalRequestHold := #sx_RightExternalRequestHold720,
	                                     ix_ResetEnergySave := FALSE,
	                                     qUDT_HMIStatus => #iqUDT_WorkstationStatus."720".Conveyor,
	                                     qUDT_Status => #iqUDT_WorkstationCommonStatus."720",
	                                     iqUDT_EquipmentControl := #iqUDT_EquipmentControl,
	                                     iqUDT_ConveyorCommand := #iqUDT_WorkstationCommands."720".Conveyor,
	                                     iqUDT_ConveyorInterface := #sUDT_Interface720,
	                                     iqUDT_HandShakeUp := #sUDT_Handshake710,
	                                     iqUDT_HandShake := #sUDT_Handshake720,
	                                     iqUDT_Statistics := #iqUDT_WorkstationStatistics."720".Conveyor);
	                END_REGION

	                REGION MCO

	                    #sFB_MCOConveyLinxAixController720(iUDT_AixConfig := #iUDT_Configuration."720".MCO_M01,
	                                                       iUDT_AixInputsModule := #iUDT_MotorInput710,
	                                                       ix_24vOk := #ix_24vOk,
	                                                       ix_SimulationModeActive := "DB_Memory".Simulation,
	                                                       ii_MotorPositionId := 2,
	                                                       qUDT_HMIStatus => #iqUDT_WorkstationStatus."720".MCO_M01,
	                                                       iqUDT_AixOutputsModule := #iqUDT_MotorOutput710,
	                                                       iqUDT_ConveyorInterface := #sUDT_Interface720,
	                                                       iqUDT_MCOStatistics := #iqUDT_WorkstationStatistics."720".MCO_M01);
	                END_REGION

	            END_REGION

	            REGION 730

	                REGION Displacement

	                    #sFB_Displacement730(#sUDT_Interface730);

	                END_REGION

	                REGION EOS
	                    #sFB_PEC730(ix_PEC := NOT #iUDT_MotorInput730.AllSensorPortInputs.LeftSensor,
	                                iUDT_PECConfiguration := #iUDT_Configuration."730".PEC_Eos,
	                                qx_PECFiltered => #tx_dummy,
	                                qUDT_HMIStatus => #iqUDT_WorkstationStatus."730".PEC_EoS,
	                                iqUDT_ConveyorInterface := #sUDT_Interface730,
	                                iqUDT_PECStatistics := #iqUDT_WorkstationStatistics."730".PEC_EoS);


	                END_REGION

	                REGION Conveyor

